FUNCTION_BLOCK FB_SignalHandling IMPLEMENTS I_SignalHandling
VAR_INPUT
	bInputSignal				AT %I*		:		BOOL;			// Hardware input signal from sensor
END_VAR
VAR_OUTPUT
	bOutputSignal				AT %Q*		:		BOOL;			// Hardware output singnal, e.g. delayed, inverted
END_VAR
VAR
	bEnableInputLocal						:		BOOL;			// Enabling processing of input signal
END_VAR

// ===========================================================================
;
// ===========================================================================

METHOD Enable
VAR_INPUT
	bEnable	: BOOL;
END_VAR
bEnableInputLocal := bEnable;
END_METHOD

METHOD SetOutput

	bOutputSignal		:=		bInputSignal AND bEnableInputLocal;
END_METHOD

END_FUNCTION_BLOCK

(* stored: Version 1.1.0.1, ProductVersion 3.1.4024.15
   POU FB_SignalHandling: Id {5ca51423-c788-41b2-96e4-6aec8675dedb}, SpecialFunc None
   Method Enable: Id {d18cf4c8-bdef-4c99-a0a6-91558625e0cd}
   Method SetOutput: Id {dd8d0faa-b781-400a-acd3-32349b3c8242} *)
